TYPE T_Syntax_Types :
    STRUCT
        nSubrange   : INT(0..100) := 50;
        aMatrix     : ARRAY[1..3, 1..3] OF REAL;
        sCustomText : STRING(255);
    END_STRUCT
END_TYPE

(* stored: Version 1.1.0.1, ProductVersion 3.1.4024.16
   DUT T_Syntax_Types: Id {10e3c610-3666-4282-840d-2574b4694439} *)
